(* IEC 61131-3 sources: RetroPLC_IDE/RetroPLC.Shell/ProjectFiles/POUs/Functions, 1 file *)

(* ---- Scale.st ---- *)
FUNCTION Scale : REAL
VAR_INPUT
    RawValue : INT;
    RawMinimum : INT;
    RawMaximum : INT;
    EngineeringMinimum : REAL;
    EngineeringMaximum : REAL;
END_VAR

Scale := EngineeringMinimum
    + INT_TO_REAL(RawValue - RawMinimum)
    * (EngineeringMaximum - EngineeringMinimum)
    / INT_TO_REAL(RawMaximum - RawMinimum);
END_FUNCTION
